Fanuc KAREL source: kd00044.KL

-- PROVISIONAL review KL for V1013-1; original PC SHA256 5e60859708bf1ef0e52024e539b9943270c00bd11571c32a637be3146362a707
-- Incomplete behavior may be omitted. Consult companion uncertainty JSON. Do not deploy.
PROGRAM KD00044
%NOLOCKGROUP
VAR
  I : INTEGER
  J : INTEGER
  B : BOOLEAN
  R : REAL
  S : STRING[80]
-- UNRESOLVED_DECL G type=00011e
BEGIN
  -- UNRESOLVED_PC offsets 5-12; opcodes 9D,23
  -- UNRESOLVED_PC offsets 17-21; opcodes 7F
END KD00044
